// TwinCAT 3 PLC project lcls_dream_motion
// Title: lcls-dream-motion
// Company: SLAC
// ProjectVersion: 1.0.0
// ProgramVersion: 3.1.4026.17
// libraries:
//   LCLS General, * (SLAC)
//   lcls-twincat-motion, * (SLAC)
//   PMPS, * (SLAC - LCLS)
//   Tc2_MC2, * (Beckhoff Automation GmbH)
//   Tc2_Standard, * (Beckhoff Automation GmbH)
//   Tc2_System, * (Beckhoff Automation GmbH)
//   Tc3_IPCDiag, * (Beckhoff Automation GmbH)
//   Tc3_Module, * (Beckhoff Automation GmbH)
// project tree:
//   DUTs/ ENUM_AxisStates.TcDUT
//   GVLs/ GVL_EPS.TcGVL, GVL_PLC_Interfaces.TcGVL, GVL_PMPS.TcGVL, Main.TcGVL
//   / PlcTask.TcTTO
//   POUs/ PRG_SMARACT.TcPOU, PRG_CoilMovers.TcPOU, PRG_GasJetPointing.TcPOU, PRG_PLC_tasks.TcPOU, PRG_GasNozzleXYZ.TcPOU, PRG_MainChamber.TcPOU
// real-time tasks:
//   TASK PlcTask: cycle T#10ms, priority 20, ADS port 350
// motion (NC):
//   TASK NC-Task 1: cycle T#2ms, priority 4, ADS port 501
//   TASK NC- Task 1 SVB: cycle T#10ms, priority 8, ADS port 511
//   AXIS M1 -MMS-Y (id 1)
//     Dynamic: AccelerationMaximum=250, DecelerationMaximum=250, Acceleration=250, Deceleration=250, DelayTime=0.008
//     Velo: Maximum=2.5
//     OtherSettings: AllowMotionCmdToSlave=true
//     encoder EncType=29
//       EncPara: ScaleFactorNumerator=5e-05, MaxCount=#xffffffff
//         SoftEndMinControl: Range=98.55
//         SoftEndMaxControl: Range=98.73
//         Inc: RefSoftSyncMask=#x0000ffff
//     drive DrvType=24
//       Analog: VeloReferenz=2.5, ScaleFactorActTorque=0.1
//       TimeComp: TaskDelayCycles=1
//     controller CtrType=2
//       CtrPara: PriorControlFactor=1
//         PosDiffControl: Range=0.3
//         PID: PosKp=0.1, PosExtVelo=0.2, DeadBandPosition=0.1
//         Observer: BandWidth=20
//   AXIS M6_GSJN-MMS-X (id 6)
//     Dynamic: AccelerationMaximum=500, DecelerationMaximum=500, Acceleration=50, Deceleration=50, Jerk=500
//     Velo: Maximum=5
//     PositionAreaControl: Range=0.0015625
//     TargetPosControl: Range=0.0015625
//     OtherSettings: AllowMotionCmdToSlave=true
//     encoder EncType=29
//       EncPara: ScaleFactorNumerator=0.000244140625, Offset=-33543453.28, MaxCount=#xffffffff, MaxCountHighDWord=#x0000001f, ReferenceSystem=1
//         FilterTime: TVelo=0.1
//         SoftEndMinControl: Enable=true, Range=-13.5
//         SoftEndMaxControl: Enable=true, Range=11.5
//         Inc: RefSoftSyncMask=#x0000ffff
//     drive DrvType=24
//       Analog: VeloReferenz=12.5, ScaleFactorActTorque=0.1
//       TimeComp: TaskDelayCycles=1
//     controller CtrType=1
//       CtrPara: PriorControlFactor=1
//         PosDiffControl: Range=0.1
//         Observer: BandWidth=20
//   AXIS M8_GSJN-MMS-Z (id 8)
//     Dynamic: AccelerationMaximum=500, DecelerationMaximum=500, Acceleration=50, Deceleration=50, Jerk=500
//     Velo: Maximum=5
//     PositionAreaControl: Range=0.002
//     TargetPosControl: Range=0.002, Time=0.1
//     OtherSettings: AllowMotionCmdToSlave=true, NoMotionFilterTime=0.05
//     encoder EncType=29
//       EncPara: ScaleFactorNumerator=0.000244140625, Offset=-33543954.59, MaxCount=#xffffffff, MaxCountHighDWord=#x0000001f, ReferenceSystem=1
//         SoftEndMinControl: Enable=true, Range=-3.5
//         SoftEndMaxControl: Enable=true, Range=4
//         Inc: RefSoftSyncMask=#x0000ffff
//     drive DrvType=24
//       Analog: VeloReferenz=12.5, ScaleFactorActTorque=0.1
//       TimeComp: TaskDelayCycles=1
//     controller CtrType=2
//       CtrPara: PriorControlFactor=1
//         PosDiffControl: Range=0.1
//         PID: PosKp=5, PosExtKp=1, DeadBandPosition=0.001
//         Observer: BandWidth=20
//   AXIS M7_GSJN-MMS-Y (id 7)
//     Dynamic: AccelerationMaximum=500, DecelerationMaximum=500, Acceleration=50, Deceleration=50, Jerk=500
//     Velo: SlowManual=1, FastManual=2, Maximum=5.08
//     PositionAreaControl: Range=0.00127
//     TargetPosControl: Range=0.00127
//     OtherSettings: AllowMotionCmdToSlave=true, PulseDistancePos=1, PulseDistanceNeg=1
//     encoder EncType=29
//       EncPara: ScaleFactorNumerator=0.000244140625, Offset=-33550977.0786, MaxCount=#xffffffff, MaxCountHighDWord=#x0000001f, ReferenceSystem=1
//         SoftEndMinControl: Enable=true, Range=-71.06
//         SoftEndMaxControl: Enable=true, Range=0.5
//         Inc: RefSoftSyncMask=#x0000ffff
//     drive DrvType=24
//       Analog: VeloReferenz=5.08, ScaleFactorActTorque=0.1
//       TimeComp: TaskDelayCycles=1
//     controller CtrType=1
//       CtrPara: PriorControlFactor=1
//         PosDiffControl: Range=0.1
//         PID: PosKp=3
//         Observer: BandWidth=20
//   AXIS M10_DREAM_DGPD_MMT_X (id 10)
//     Dynamic: AccelerationMaximum=10, DecelerationMaximum=10, Acceleration=2.51748, Deceleration=2.51748, Jerk=9.32019
//     Velo: RefSearch=0.5, RefSync=0.4, SlowManual=0.2, FastManual=0.2, Maximum=1
//     PositionAreaControl: Range=0.005
//     TargetPosControl: Enable=false
//     OtherSettings: AllowMotionCmdToSlave=true, PulseDistancePos=0.01, PulseDistanceNeg=0.01
//     encoder EncType=19
//       EncPara: ScaleFactorNumerator=1e-06, MaxCount=#xffffffff
//     drive DrvType=16
//       DrvPara: MaxCount=#xffffffff, DriveControlDWord=#x00020100
//         Analog: VeloReferenz=1, TorqueSetpointScale=10, ScaleFactorActTorque=0.1
//         TimeComp: TaskDelayCycles=1
//     controller CtrType=1
//       CtrPara: PriorControlFactor=1
//         PosDiffControl: Range=0.05
//         Observer: BandWidth=20
//   AXIS M11_DREAM_DGPD_MMT_RET (id 11)
//     Dynamic: AccelerationMaximum=10, DecelerationMaximum=10, Acceleration=2.51748, Deceleration=2.51748, Jerk=9.32019
//     Velo: RefSearch=0.5, RefSync=0.4, SlowManual=0.2, FastManual=0.2, Maximum=1
//     PositionAreaControl: Range=0.005
//     TargetPosControl: Enable=false
//     OtherSettings: AllowMotionCmdToSlave=true, PulseDistancePos=0.01, PulseDistanceNeg=0.01
//     encoder EncType=19
//       EncPara: ScaleFactorNumerator=1e-06, MaxCount=#xffffffff
//     drive DrvType=16
//       DrvPara: MaxCount=#xffffffff, DriveControlDWord=#x00020100
//         Analog: VeloReferenz=1, TorqueSetpointScale=10, ScaleFactorActTorque=0.1
//         TimeComp: TaskDelayCycles=1
//     controller CtrType=1
//       CtrPara: PriorControlFactor=1
//         PosDiffControl: Range=0.05
//         Observer: BandWidth=20
//   AXIS M9_DREAM_DGPD_MMT_Y (id 9)
//     Dynamic: AccelerationMaximum=10, DecelerationMaximum=10, Acceleration=2.51748, Deceleration=2.51748, Jerk=9.32019
//     Velo: RefSearch=0.5, RefSync=0.4, SlowManual=0.2, FastManual=0.2, Maximum=1
//     PositionAreaControl: Range=0.005
//     TargetPosControl: Enable=false
//     OtherSettings: AllowMotionCmdToSlave=true, PulseDistancePos=0.01, PulseDistanceNeg=0.01
//     encoder EncType=19
//       EncPara: ScaleFactorNumerator=1e-06, MaxCount=#xffffffff
//     drive DrvType=16
//       DrvPara: MaxCount=#xffffffff, DriveControlDWord=#x00020100
//         Analog: VeloReferenz=1, TorqueSetpointScale=10, ScaleFactorActTorque=0.1
//         TimeComp: TaskDelayCycles=1
//     controller CtrType=1
//       CtrPara: PriorControlFactor=1
//         PosDiffControl: Range=0.05
//         Observer: BandWidth=20
//   AXIS M2 - Coil Roll (id 2)
//     Dynamic: AccelerationMaximum=1600, DecelerationMaximum=1600, Acceleration=1600, Deceleration=1600
//     Velo: Maximum=16
//     OtherSettings: AllowMotionCmdToSlave=true
//     encoder EncType=7
//       EncPara: ScaleFactorNumerator=0.004566812625, Offset=-59.42, MaxCount=#x0000ffff, ReferenceSystem=1
//         SoftEndMinControl: Enable=true, Range=-53.06
//         SoftEndMaxControl: Enable=true, Range=75.44
//         Inc: RefSoftSyncMask=#x0000ffff
//     drive DrvType=24
//       Analog: VeloReferenz=15.875, ScaleFactorActTorque=0.1
//       TimeComp: TaskDelayCycles=1
//     controller CtrType=1
//       CtrPara: PriorControlFactor=1
//         PosDiffControl: Range=1
//         Observer: BandWidth=20
//   AXIS M3 - Coil Yaw (id 3)
//     Dynamic: AccelerationMaximum=1600, DecelerationMaximum=1600
//     Velo: Maximum=16
//     OtherSettings: AllowMotionCmdToSlave=true
//     encoder EncType=7
//       EncPara: ScaleFactorNumerator=0.004566812625, Offset=-137.15, MaxCount=#x0000ffff, ReferenceSystem=1
//         SoftEndMinControl: Enable=true, Range=-3.65
//         SoftEndMaxControl: Enable=true, Range=6.35
//         Inc: RefSoftSyncMask=#x0000ffff
//     drive DrvType=24
//       Analog: VeloReferenz=15.875, ScaleFactorActTorque=0.1
//       TimeComp: TaskDelayCycles=1
//     controller CtrType=1
//       CtrPara: PriorControlFactor=1
//         PosDiffControl: Range=0.75
//         PID: PosKp=1.1
//         Observer: BandWidth=20
//   AXIS M4 - GSJP X (id 4)
//     Velo: Maximum=15.875
//     OtherSettings: AllowMotionCmdToSlave=true
//     encoder EncType=7
//       EncPara: ScaleFactorNumerator=0.0016164154, Offset=-19.9643, MaxCount=#x0000ffff, ReferenceSystem=1
//         SoftEndMinControl: Enable=true, Range=-1
//         SoftEndMaxControl: Enable=true, Range=1
//         Inc: RefSoftSyncMask=#x0000ffff
//     drive DrvType=24
//       Analog: VeloReferenz=15.875, ScaleFactorActTorque=0.1
//       TimeComp: TaskDelayCycles=1
//     controller CtrType=1
//       CtrPara: PriorControlFactor=1
//         PosDiffControl: Range=1
//         Observer: BandWidth=20
//   AXIS M5 - GSJP Z (id 5)
//     Dynamic: AccelerationMaximum=15, DecelerationMaximum=15, Acceleration=15, Deceleration=15
//     Velo: Maximum=16
//     OtherSettings: AllowMotionCmdToSlave=true
//     encoder EncType=7
//       EncPara: ScaleFactorNumerator=0.0016164154, Offset=-19.49, MaxCount=#x0000ffff, ReferenceSystem=1
//         SoftEndMinControl: Enable=true, Range=-1
//         SoftEndMaxControl: Enable=true, Range=1
//         Inc: RefSoftSyncMask=#x0000ffff
//     drive DrvType=24
//       DrvPara: Inverse=true
//         Analog: VeloReferenz=15.875, ScaleFactorActTorque=0.1
//         TimeComp: TaskDelayCycles=1
//     controller CtrType=1
//       CtrPara: PriorControlFactor=1
//         PosDiffControl: Range=1.5
//         Observer: BandWidth=20
// I/O:
//   DEVICE Device 1 (EtherCAT), AmsNetId 172.21.132.145.2.1
//     B940_009_R19_DRL_02_E0_EK1200 [EK1200-5000 EtherCAT Power supply (2A E-Bus)]
//       R19_DRL_02_EL2202
//       R19_DRL_02_E2_EL6070
//       R19_DRL_02_E3_EL6695 [EL6695 EtherCAT Bridge terminal (Primary)]
//       R19_DRL_02_E4_EK1122 [EK1122 2 port EtherCAT junction]
//         K4S08_DRL_05_E0_EK1100 [EK1100 EtherCAT Coupler (2A E-Bus)]
//           DRL_05_EL7047_E1 [EL7047 1Ch. Stepper motor output stage (50V, 5A)]
//           DRL_05_EL5042_E2 [EL5042 2Ch. BiSS-C Encoder]
//           DRL_05_EL7047_E3 [EL7047 1Ch. Stepper motor output stage (50V, 5A)]
//           DRL_05_EL7047_E4 [EL7047 1Ch. Stepper motor output stage (50V, 5A)]
//           DRL_05_EL3064_E5
//           DRL_05_EL7047_E6 [EL7047 1Ch. Stepper motor output stage (50V, 5A)]
//           DRL_05_EL7047_E7 [EL7047 1Ch. Stepper motor output stage (50V, 5A)]
//           DRL_05_EL7047_E9 [EL7047 1Ch. Stepper motor output stage (50V, 5A)]
//           DRL_05_EL7047_E10 [EL7047 1Ch. Stepper motor output stage (50V, 5A)]
//           DRL_05_EL5042_E11 [EL5042 2Ch. BiSS-C Encoder]
//           DRL_05_EL7047_E12 [EL7047 1Ch. Stepper motor output stage (50V, 5A)]
//           DRL_05_EL9011 [EL9011 End Terminal]
//         Term 35 (EK1100) [EK1100 EtherCAT Coupler (2A E-Bus)]
//           B950-100H1-R02-PNL-01_E1 [EL2624 4Ch. Relay Output, NO (125V AC / 30V DC)]
//           B950-100H1-R02-PNL-01_E2 [EL1002 2Ch. Dig. Input 24V, 3ms]
//           Term 41 (EL9011) [EL9011 End Terminal]
//         TMO-DREAM-SMARACT-03 [MCS2-3C] (disabled)
//           modules: DREAM:DGPD:MMT:Y, DREAM:DGPD:MMT:X, DREAM:DGPD:MMT:RET
//       B940_009_R19_DRL_02_E5_ EL6695 [EL6695 EtherCAT Bridge terminal (Primary)]
//       Term 42 (EL9011) [EL9011 End Terminal]
// variable links:
//   (this object) <-> Device 1 (EtherCAT)/B940_009_R19_DRL_02_E0_EK1200/R19_DRL_02_E4_EK1122/K4S08_DRL_05_E0_EK1100/DRL_05_EL5042_E2
//     Enc/Inputs/In/nComState @bit 1 <-> WcState/InputToggle
//     Enc/Inputs/In/nComState <-> WcState/WcState
//     Enc/Inputs/In/nDataIn1 <-> FB Inputs Channel 1/Position
//     Enc/Inputs/In/nDataIn1 <-> FB Inputs Channel 2/Position
//     Enc/Inputs/In/nState1 @bit 12 <-> FB Inputs Channel 1/Status/Diag
//     Enc/Inputs/In/nState1 @bit 12 <-> FB Inputs Channel 2/Status/Diag
//     Enc/Inputs/In/nState1 @bit 1 <-> FB Inputs Channel 1/Status/Error
//     Enc/Inputs/In/nState1 @bit 1 <-> FB Inputs Channel 2/Status/Error
//     Enc/Inputs/In/nState1 @bit 14 <-> FB Inputs Channel 1/Status/Input cycle counter
//     Enc/Inputs/In/nState1 @bit 14 <-> FB Inputs Channel 2/Status/Input cycle counter
//     Enc/Inputs/In/nState1 @bit 2 <-> FB Inputs Channel 1/Status/Ready
//     Enc/Inputs/In/nState1 @bit 2 <-> FB Inputs Channel 2/Status/Ready
//     Enc/Inputs/In/nState1 @bit 13 <-> FB Inputs Channel 1/Status/TxPDO State
//     Enc/Inputs/In/nState1 @bit 13 <-> FB Inputs Channel 2/Status/TxPDO State
//     Enc/Inputs/In/nState1 <-> FB Inputs Channel 1/Status/Warning
//     Enc/Inputs/In/nState1 <-> FB Inputs Channel 2/Status/Warning
//   (this object) <-> Device 1 (EtherCAT)/B940_009_R19_DRL_02_E0_EK1200/R19_DRL_02_E4_EK1122/K4S08_DRL_05_E0_EK1100/DRL_05_EL7047_E1
//     Drive/Inputs/In/nState1 @bit 3 <-> STM Status/Status/Error
//     Drive/Inputs/In/nState1 @bit 7 <-> STM Status/Status/Motor stall
//     Drive/Inputs/In/nState1 @bit 5 <-> STM Status/Status/Moving negative
//     Drive/Inputs/In/nState1 @bit 4 <-> STM Status/Status/Moving positive
//     Drive/Inputs/In/nState1 @bit 1 <-> STM Status/Status/Ready
//     Drive/Inputs/In/nState1 <-> STM Status/Status/Ready to enable
//     Drive/Inputs/In/nState1 @bit 6 <-> STM Status/Status/Torque reduced
//     Drive/Inputs/In/nState1 @bit 2 <-> STM Status/Status/Warning
//     Drive/Inputs/In/nState2 @bit 3 <-> STM Status/Status/Digital input 1
//     Drive/Inputs/In/nState2 @bit 4 <-> STM Status/Status/Digital input 2
//     Drive/Inputs/In/nState2 @bit 5 <-> STM Status/Status/Sync error
//     Drive/Inputs/In/nState2 @bit 7 <-> STM Status/Status/TxPDO Toggle
//     Drive/Inputs/In/nState4 @bit 1 <-> WcState/InputToggle
//     Drive/Inputs/In/nState4 <-> WcState/WcState
//     Drive/Outputs/Out/nCtrl1 <-> STM Control/Control/Enable
//     Drive/Outputs/Out/nCtrl1 @bit 2 <-> STM Control/Control/Reduce torque
//     Drive/Outputs/Out/nCtrl1 @bit 1 <-> STM Control/Control/Reset
//     Drive/Outputs/Out/nCtrl2 @bit 3 <-> STM Control/Control/Digital output 1
//     Drive/Outputs/Out/nDataOut2[0] <-> STM Velocity/Velocity
//   (this object) <-> Device 1 (EtherCAT)/B940_009_R19_DRL_02_E0_EK1200/R19_DRL_02_E4_EK1122/K4S08_DRL_05_E0_EK1100/DRL_05_EL7047_E9
//     Drive/Inputs/In/nState1 @bit 3 <-> STM Status/Status/Error
//     Drive/Inputs/In/nState1 @bit 7 <-> STM Status/Status/Motor stall
//     Drive/Inputs/In/nState1 @bit 5 <-> STM Status/Status/Moving negative
//     Drive/Inputs/In/nState1 @bit 4 <-> STM Status/Status/Moving positive
//     Drive/Inputs/In/nState1 @bit 1 <-> STM Status/Status/Ready
//     Drive/Inputs/In/nState1 <-> STM Status/Status/Ready to enable
//     Drive/Inputs/In/nState1 @bit 6 <-> STM Status/Status/Torque reduced
//     Drive/Inputs/In/nState1 @bit 2 <-> STM Status/Status/Warning
//     Drive/Inputs/In/nState2 @bit 3 <-> STM Status/Status/Digital input 1
//     Drive/Inputs/In/nState2 @bit 4 <-> STM Status/Status/Digital input 2
//     Drive/Inputs/In/nState2 @bit 5 <-> STM Status/Status/Sync error
//     Drive/Inputs/In/nState2 @bit 7 <-> STM Status/Status/TxPDO Toggle
//     Drive/Inputs/In/nState4 @bit 1 <-> WcState/InputToggle
//     Drive/Inputs/In/nState4 <-> WcState/WcState
//     Drive/Outputs/Out/nCtrl1 <-> STM Control/Control/Enable
//     Drive/Outputs/Out/nCtrl1 @bit 2 <-> STM Control/Control/Reduce torque
//     Drive/Outputs/Out/nCtrl1 @bit 1 <-> STM Control/Control/Reset
//     Drive/Outputs/Out/nCtrl2 @bit 3 <-> STM Control/Control/Digital output 1
//     Drive/Outputs/Out/nDataOut2[0] <-> STM Velocity/Velocity
//   (this object) <-> Device 1 (EtherCAT)/B940_009_R19_DRL_02_E0_EK1200/R19_DRL_02_E4_EK1122/K4S08_DRL_05_E0_EK1100/DRL_05_EL5042_E11
//     Enc/Inputs/In/nComState @bit 1 <-> WcState/InputToggle
//     Enc/Inputs/In/nComState <-> WcState/WcState
//     Enc/Inputs/In/nDataIn1 <-> FB Inputs Channel 2/Position
//     Enc/Inputs/In/nDataIn1 <-> FB Inputs Channel 1/Position
//     Enc/Inputs/In/nState1 @bit 12 <-> FB Inputs Channel 2/Status/Diag
//     Enc/Inputs/In/nState1 @bit 12 <-> FB Inputs Channel 1/Status/Diag
//     Enc/Inputs/In/nState1 @bit 1 <-> FB Inputs Channel 2/Status/Error
//     Enc/Inputs/In/nState1 @bit 1 <-> FB Inputs Channel 1/Status/Error
//     Enc/Inputs/In/nState1 @bit 14 <-> FB Inputs Channel 2/Status/Input cycle counter
//     Enc/Inputs/In/nState1 @bit 14 <-> FB Inputs Channel 1/Status/Input cycle counter
//     Enc/Inputs/In/nState1 @bit 2 <-> FB Inputs Channel 2/Status/Ready
//     Enc/Inputs/In/nState1 @bit 2 <-> FB Inputs Channel 1/Status/Ready
//     Enc/Inputs/In/nState1 @bit 13 <-> FB Inputs Channel 2/Status/TxPDO State
//     Enc/Inputs/In/nState1 @bit 13 <-> FB Inputs Channel 1/Status/TxPDO State
//     Enc/Inputs/In/nState1 <-> FB Inputs Channel 2/Status/Warning
//     Enc/Inputs/In/nState1 <-> FB Inputs Channel 1/Status/Warning
//   (this object) <-> Device 1 (EtherCAT)/B940_009_R19_DRL_02_E0_EK1200/R19_DRL_02_E4_EK1122/K4S08_DRL_05_E0_EK1100/DRL_05_EL7047_E12
//     Drive/Inputs/In/nState1 @bit 3 <-> STM Status/Status/Error
//     Drive/Inputs/In/nState1 @bit 7 <-> STM Status/Status/Motor stall
//     Drive/Inputs/In/nState1 @bit 5 <-> STM Status/Status/Moving negative
//     Drive/Inputs/In/nState1 @bit 4 <-> STM Status/Status/Moving positive
//     Drive/Inputs/In/nState1 @bit 1 <-> STM Status/Status/Ready
//     Drive/Inputs/In/nState1 <-> STM Status/Status/Ready to enable
//     Drive/Inputs/In/nState1 @bit 6 <-> STM Status/Status/Torque reduced
//     Drive/Inputs/In/nState1 @bit 2 <-> STM Status/Status/Warning
//     Drive/Inputs/In/nState2 @bit 3 <-> STM Status/Status/Digital input 1
//     Drive/Inputs/In/nState2 @bit 4 <-> STM Status/Status/Digital input 2
//     Drive/Inputs/In/nState2 @bit 5 <-> STM Status/Status/Sync error
//     Drive/Inputs/In/nState2 @bit 7 <-> STM Status/Status/TxPDO Toggle
//     Drive/Inputs/In/nState4 @bit 1 <-> WcState/InputToggle
//     Drive/Inputs/In/nState4 <-> WcState/WcState
//     Drive/Outputs/Out/nCtrl1 <-> STM Control/Control/Enable
//     Drive/Outputs/Out/nCtrl1 @bit 2 <-> STM Control/Control/Reduce torque
//     Drive/Outputs/Out/nCtrl1 @bit 1 <-> STM Control/Control/Reset
//     Drive/Outputs/Out/nCtrl2 @bit 3 <-> STM Control/Control/Digital output 1
//     Drive/Outputs/Out/nDataOut2[0] <-> STM Velocity/Velocity
//   (this object) <-> Device 1 (EtherCAT)/B940_009_R19_DRL_02_E0_EK1200/R19_DRL_02_E4_EK1122/K4S08_DRL_05_E0_EK1100/DRL_05_EL7047_E10
//     Drive/Inputs/In/nState1 @bit 3 <-> STM Status/Status/Error
//     Drive/Inputs/In/nState1 @bit 7 <-> STM Status/Status/Motor stall
//     Drive/Inputs/In/nState1 @bit 5 <-> STM Status/Status/Moving negative
//     Drive/Inputs/In/nState1 @bit 4 <-> STM Status/Status/Moving positive
//     Drive/Inputs/In/nState1 @bit 1 <-> STM Status/Status/Ready
//     Drive/Inputs/In/nState1 <-> STM Status/Status/Ready to enable
//     Drive/Inputs/In/nState1 @bit 6 <-> STM Status/Status/Torque reduced
//     Drive/Inputs/In/nState1 @bit 2 <-> STM Status/Status/Warning
//     Drive/Inputs/In/nState2 @bit 3 <-> STM Status/Status/Digital input 1
//     Drive/Inputs/In/nState2 @bit 4 <-> STM Status/Status/Digital input 2
//     Drive/Inputs/In/nState2 @bit 5 <-> STM Status/Status/Sync error
//     Drive/Inputs/In/nState2 @bit 7 <-> STM Status/Status/TxPDO Toggle
//     Drive/Inputs/In/nState4 @bit 1 <-> WcState/InputToggle
//     Drive/Inputs/In/nState4 <-> WcState/WcState
//     Drive/Outputs/Out/nCtrl1 <-> STM Control/Control/Enable
//     Drive/Outputs/Out/nCtrl1 @bit 2 <-> STM Control/Control/Reduce torque
//     Drive/Outputs/Out/nCtrl1 @bit 1 <-> STM Control/Control/Reset
//     Drive/Outputs/Out/nCtrl2 @bit 3 <-> STM Control/Control/Digital output 1
//     Drive/Outputs/Out/nDataOut2[0] <-> STM Velocity/Velocity
//   (this object) <-> Device 1 (EtherCAT)/B940_009_R19_DRL_02_E0_EK1200/R19_DRL_02_E4_EK1122/TMO-DREAM-SMARACT-03
//     Drive/Inputs/In/nDataIn1 <-> DREAM:DGPD:MMT:X/mode/status/pos/fError TxPDO/Following Error Actual Value
//     Drive/Inputs/In/nState1 <-> DREAM:DGPD:MMT:X/mode/status/pos/fError TxPDO/Status Word
//     Drive/Inputs/In/nState2 <-> DREAM:DGPD:MMT:X/mode/status/pos/fError TxPDO/Status Word @bit 8
//     Drive/Inputs/In/nState4 @bit 1 <-> WcState/InputToggle
//     Drive/Inputs/In/nState4 <-> WcState/WcState
//     Drive/Inputs/In/nState5 <-> DREAM:DGPD:MMT:X/mode/status/pos/fError TxPDO/Modes of Operation Display
//     Drive/Outputs/Out/nDataOut1 <-> DREAM:DGPD:MMT:X/ctl/mode/pos RxPDO/Target Position
//     Enc/Inputs/In/nDataIn1 <-> DREAM:DGPD:MMT:X/mode/status/pos/fError TxPDO/Position Actual Value
//     Enc/Inputs/In/nState4 @bit 1 <-> WcState/InputToggle
//     Enc/Inputs/In/nState4 <-> WcState/WcState
//     Drive/Inputs/In/nDataIn1 <-> DREAM:DGPD:MMT:RET/mode/status/pos/fError TxPDO/Following Error Actual Value
//     Drive/Inputs/In/nState1 <-> DREAM:DGPD:MMT:RET/mode/status/pos/fError TxPDO/Status Word
//     Drive/Inputs/In/nState2 <-> DREAM:DGPD:MMT:RET/mode/status/pos/fError TxPDO/Status Word @bit 8
//     Drive/Inputs/In/nState5 <-> DREAM:DGPD:MMT:RET/mode/status/pos/fError TxPDO/Modes of Operation Display
//     Drive/Outputs/Out/nDataOut1 <-> DREAM:DGPD:MMT:RET/ctl/mode/pos RxPDO/Target Position
//     Enc/Inputs/In/nDataIn1 <-> DREAM:DGPD:MMT:RET/mode/status/pos/fError TxPDO/Position Actual Value
//     Drive/Inputs/In/nDataIn1 <-> DREAM:DGPD:MMT:Y/mode/status/pos/fError TxPDO/Following Error Actual Value
//     Drive/Inputs/In/nState1 <-> DREAM:DGPD:MMT:Y/mode/status/pos/fError TxPDO/Status Word
//     Drive/Inputs/In/nState2 <-> DREAM:DGPD:MMT:Y/mode/status/pos/fError TxPDO/Status Word @bit 8
//     Drive/Inputs/In/nState5 <-> DREAM:DGPD:MMT:Y/mode/status/pos/fError TxPDO/Modes of Operation Display
//     Drive/Outputs/Out/nDataOut1 <-> DREAM:DGPD:MMT:Y/ctl/mode/pos RxPDO/Target Position
//     Enc/Inputs/In/nDataIn1 <-> DREAM:DGPD:MMT:Y/mode/status/pos/fError TxPDO/Position Actual Value
//   (this object) <-> Device 1 (EtherCAT)/B940_009_R19_DRL_02_E0_EK1200/R19_DRL_02_E4_EK1122/K4S08_DRL_05_E0_EK1100/DRL_05_EL3064_E5
//     Enc/Inputs/In/nDataIn1[0] <-> AI Standard Channel {1..4}/Value  (4 links)
//     Enc/Inputs/In/nState4 @bit 1 <-> WcState/InputToggle
//     Enc/Inputs/In/nState4 <-> WcState/WcState
//   (this object) <-> Device 1 (EtherCAT)/B940_009_R19_DRL_02_E0_EK1200/R19_DRL_02_E4_EK1122/K4S08_DRL_05_E0_EK1100/DRL_05_EL7047_E3
//     Drive/Inputs/In/nState1 @bit 3 <-> STM Status/Status/Error
//     Drive/Inputs/In/nState1 @bit 7 <-> STM Status/Status/Motor stall
//     Drive/Inputs/In/nState1 @bit 5 <-> STM Status/Status/Moving negative
//     Drive/Inputs/In/nState1 @bit 4 <-> STM Status/Status/Moving positive
//     Drive/Inputs/In/nState1 @bit 1 <-> STM Status/Status/Ready
//     Drive/Inputs/In/nState1 <-> STM Status/Status/Ready to enable
//     Drive/Inputs/In/nState1 @bit 6 <-> STM Status/Status/Torque reduced
//     Drive/Inputs/In/nState1 @bit 2 <-> STM Status/Status/Warning
//     Drive/Inputs/In/nState2 @bit 3 <-> STM Status/Status/Digital input 1
//     Drive/Inputs/In/nState2 @bit 4 <-> STM Status/Status/Digital input 2
//     Drive/Inputs/In/nState2 @bit 5 <-> STM Status/Status/Sync error
//     Drive/Inputs/In/nState2 @bit 7 <-> STM Status/Status/TxPDO Toggle
//     Drive/Inputs/In/nState4 @bit 1 <-> WcState/InputToggle
//     Drive/Inputs/In/nState4 <-> WcState/WcState
//     Drive/Outputs/Out/nCtrl1 <-> STM Control/Control/Enable
//     Drive/Outputs/Out/nCtrl1 @bit 2 <-> STM Control/Control/Reduce torque
//     Drive/Outputs/Out/nCtrl1 @bit 1 <-> STM Control/Control/Reset
//     Drive/Outputs/Out/nCtrl2 @bit 3 <-> STM Control/Control/Digital output 1
//     Drive/Outputs/Out/nDataOut2[0] <-> STM Velocity/Velocity
//   (this object) <-> Device 1 (EtherCAT)/B940_009_R19_DRL_02_E0_EK1200/R19_DRL_02_E4_EK1122/K4S08_DRL_05_E0_EK1100/DRL_05_EL7047_E4
//     Drive/Inputs/In/nState1 @bit 3 <-> STM Status/Status/Error
//     Drive/Inputs/In/nState1 @bit 7 <-> STM Status/Status/Motor stall
//     Drive/Inputs/In/nState1 @bit 5 <-> STM Status/Status/Moving negative
//     Drive/Inputs/In/nState1 @bit 4 <-> STM Status/Status/Moving positive
//     Drive/Inputs/In/nState1 @bit 1 <-> STM Status/Status/Ready
//     Drive/Inputs/In/nState1 <-> STM Status/Status/Ready to enable
//     Drive/Inputs/In/nState1 @bit 6 <-> STM Status/Status/Torque reduced
//     Drive/Inputs/In/nState1 @bit 2 <-> STM Status/Status/Warning
//     Drive/Inputs/In/nState2 @bit 3 <-> STM Status/Status/Digital input 1
//     Drive/Inputs/In/nState2 @bit 4 <-> STM Status/Status/Digital input 2
//     Drive/Inputs/In/nState2 @bit 5 <-> STM Status/Status/Sync error
//     Drive/Inputs/In/nState2 @bit 7 <-> STM Status/Status/TxPDO Toggle
//     Drive/Inputs/In/nState4 @bit 1 <-> WcState/InputToggle
//     Drive/Inputs/In/nState4 <-> WcState/WcState
//     Drive/Outputs/Out/nCtrl1 <-> STM Control/Control/Enable
//     Drive/Outputs/Out/nCtrl1 @bit 2 <-> STM Control/Control/Reduce torque
//     Drive/Outputs/Out/nCtrl1 @bit 1 <-> STM Control/Control/Reset
//     Drive/Outputs/Out/nCtrl2 @bit 3 <-> STM Control/Control/Digital output 1
//     Drive/Outputs/Out/nDataOut2[0] <-> STM Velocity/Velocity
//   (this object) <-> Device 1 (EtherCAT)/B940_009_R19_DRL_02_E0_EK1200/R19_DRL_02_E4_EK1122/K4S08_DRL_05_E0_EK1100/DRL_05_EL7047_E6
//     Drive/Inputs/In/nState1 @bit 3 <-> STM Status/Status/Error
//     Drive/Inputs/In/nState1 @bit 7 <-> STM Status/Status/Motor stall
//     Drive/Inputs/In/nState1 @bit 5 <-> STM Status/Status/Moving negative
//     Drive/Inputs/In/nState1 @bit 4 <-> STM Status/Status/Moving positive
//     Drive/Inputs/In/nState1 @bit 1 <-> STM Status/Status/Ready
//     Drive/Inputs/In/nState1 <-> STM Status/Status/Ready to enable
//     Drive/Inputs/In/nState1 @bit 6 <-> STM Status/Status/Torque reduced
//     Drive/Inputs/In/nState1 @bit 2 <-> STM Status/Status/Warning
//     Drive/Inputs/In/nState2 @bit 3 <-> STM Status/Status/Digital input 1
//     Drive/Inputs/In/nState2 @bit 4 <-> STM Status/Status/Digital input 2
//     Drive/Inputs/In/nState2 @bit 5 <-> STM Status/Status/Sync error
//     Drive/Inputs/In/nState2 @bit 7 <-> STM Status/Status/TxPDO Toggle
//     Drive/Inputs/In/nState4 @bit 1 <-> WcState/InputToggle
//     Drive/Inputs/In/nState4 <-> WcState/WcState
//     Drive/Outputs/Out/nCtrl1 <-> STM Control/Control/Enable
//     Drive/Outputs/Out/nCtrl1 @bit 2 <-> STM Control/Control/Reduce torque
//     Drive/Outputs/Out/nCtrl1 @bit 1 <-> STM Control/Control/Reset
//     Drive/Outputs/Out/nCtrl2 @bit 3 <-> STM Control/Control/Digital output 1
//     Drive/Outputs/Out/nDataOut2[0] <-> STM Velocity/Velocity
//   (this object) <-> Device 1 (EtherCAT)/B940_009_R19_DRL_02_E0_EK1200/R19_DRL_02_E4_EK1122/K4S08_DRL_05_E0_EK1100/DRL_05_EL7047_E7
//     Drive/Inputs/In/nState1 @bit 3 <-> STM Status/Status/Error
//     Drive/Inputs/In/nState1 @bit 7 <-> STM Status/Status/Motor stall
//     Drive/Inputs/In/nState1 @bit 5 <-> STM Status/Status/Moving negative
//     Drive/Inputs/In/nState1 @bit 4 <-> STM Status/Status/Moving positive
//     Drive/Inputs/In/nState1 @bit 1 <-> STM Status/Status/Ready
//     Drive/Inputs/In/nState1 <-> STM Status/Status/Ready to enable
//     Drive/Inputs/In/nState1 @bit 6 <-> STM Status/Status/Torque reduced
//     Drive/Inputs/In/nState1 @bit 2 <-> STM Status/Status/Warning
//     Drive/Inputs/In/nState2 @bit 3 <-> STM Status/Status/Digital input 1
//     Drive/Inputs/In/nState2 @bit 4 <-> STM Status/Status/Digital input 2
//     Drive/Inputs/In/nState2 @bit 5 <-> STM Status/Status/Sync error
//     Drive/Inputs/In/nState2 @bit 7 <-> STM Status/Status/TxPDO Toggle
//     Drive/Inputs/In/nState4 @bit 1 <-> WcState/InputToggle
//     Drive/Inputs/In/nState4 <-> WcState/WcState
//     Drive/Outputs/Out/nCtrl1 <-> STM Control/Control/Enable
//     Drive/Outputs/Out/nCtrl1 @bit 2 <-> STM Control/Control/Reduce torque
//     Drive/Outputs/Out/nCtrl1 @bit 1 <-> STM Control/Control/Reset
//     Drive/Outputs/Out/nCtrl2 @bit 3 <-> STM Control/Control/Digital output 1
//     Drive/Outputs/Out/nDataOut2[0] <-> STM Velocity/Velocity
//   lcls_dream_motion Instance <-> Device 1 (EtherCAT)/B940_009_R19_DRL_02_E0_EK1200/R19_DRL_02_E4_EK1122/K4S08_DRL_05_E0_EK1100/DRL_05_EL3064_E5
//     PlcTask Inputs/Main.M{2..5}.nRawEncoderINT <-> AI Standard Channel {1..4}/Value  (4 links)
//   lcls_dream_motion Instance <-> Device 1 (EtherCAT)/B940_009_R19_DRL_02_E0_EK1200/R19_DRL_02_E4_EK1122/K4S08_DRL_05_E0_EK1100/DRL_05_EL5042_E11
//     PlcTask Inputs/Main.M7.nRawEncoderULINT <-> FB Inputs Channel 1/Position
//     PlcTask Inputs/Main.M8.nRawEncoderULINT <-> FB Inputs Channel 2/Position
//   lcls_dream_motion Instance <-> Device 1 (EtherCAT)/B940_009_R19_DRL_02_E0_EK1200/R19_DRL_02_E4_EK1122/K4S08_DRL_05_E0_EK1100/DRL_05_EL5042_E2
//     PlcTask Inputs/Main.M1.nRawEncoderULINT <-> FB Inputs Channel 1/Position
//     PlcTask Inputs/Main.M6.nRawEncoderULINT <-> FB Inputs Channel 2/Position
//   lcls_dream_motion Instance <-> Device 1 (EtherCAT)/B940_009_R19_DRL_02_E0_EK1200/R19_DRL_02_E4_EK1122/K4S08_DRL_05_E0_EK1100/DRL_05_EL7047_E1
//     PlcTask Inputs/Main.M1.bLimitBackwardEnable <-> STM Status/Status/Digital input 2
//     PlcTask Inputs/Main.M1.bLimitForwardEnable <-> STM Status/Status/Digital input 1
//   lcls_dream_motion Instance <-> Device 1 (EtherCAT)/B940_009_R19_DRL_02_E0_EK1200/R19_DRL_02_E4_EK1122/K4S08_DRL_05_E0_EK1100/DRL_05_EL7047_E10
//     PlcTask Inputs/Main.M7.bLimitBackwardEnable <-> STM Status/Status/Digital input 1
//     PlcTask Inputs/Main.M7.bLimitForwardEnable <-> STM Status/Status/Digital input 2
//   lcls_dream_motion Instance <-> Device 1 (EtherCAT)/B940_009_R19_DRL_02_E0_EK1200/R19_DRL_02_E4_EK1122/K4S08_DRL_05_E0_EK1100/DRL_05_EL7047_E12
//     PlcTask Inputs/Main.M8.bLimitBackwardEnable <-> STM Status/Status/Digital input 1
//     PlcTask Inputs/Main.M8.bLimitForwardEnable <-> STM Status/Status/Digital input 2
//   lcls_dream_motion Instance <-> Device 1 (EtherCAT)/B940_009_R19_DRL_02_E0_EK1200/R19_DRL_02_E4_EK1122/K4S08_DRL_05_E0_EK1100/DRL_05_EL7047_E3
//     PlcTask Inputs/Main.M2.bLimitBackwardEnable <-> STM Status/Status/Digital input 2
//     PlcTask Inputs/Main.M2.bLimitForwardEnable <-> STM Status/Status/Digital input 1
//   lcls_dream_motion Instance <-> Device 1 (EtherCAT)/B940_009_R19_DRL_02_E0_EK1200/R19_DRL_02_E4_EK1122/K4S08_DRL_05_E0_EK1100/DRL_05_EL7047_E4
//     PlcTask Inputs/Main.M3.bLimitBackwardEnable <-> STM Status/Status/Digital input 2
//     PlcTask Inputs/Main.M3.bLimitForwardEnable <-> STM Status/Status/Digital input 1
//   lcls_dream_motion Instance <-> Device 1 (EtherCAT)/B940_009_R19_DRL_02_E0_EK1200/R19_DRL_02_E4_EK1122/K4S08_DRL_05_E0_EK1100/DRL_05_EL7047_E6
//     PlcTask Inputs/Main.M4.bLimitBackwardEnable <-> STM Status/Status/Digital input 2
//     PlcTask Inputs/Main.M4.bLimitForwardEnable <-> STM Status/Status/Digital input 1
//   lcls_dream_motion Instance <-> Device 1 (EtherCAT)/B940_009_R19_DRL_02_E0_EK1200/R19_DRL_02_E4_EK1122/K4S08_DRL_05_E0_EK1100/DRL_05_EL7047_E7
//     PlcTask Inputs/Main.M5.bLimitBackwardEnable <-> STM Status/Status/Digital input 1
//     PlcTask Inputs/Main.M5.bLimitForwardEnable <-> STM Status/Status/Digital input 2
//   lcls_dream_motion Instance <-> Device 1 (EtherCAT)/B940_009_R19_DRL_02_E0_EK1200/R19_DRL_02_E4_EK1122/K4S08_DRL_05_E0_EK1100/DRL_05_EL7047_E9
//     PlcTask Inputs/Main.M6.bLimitBackwardEnable <-> STM Status/Status/Digital input 1
//     PlcTask Inputs/Main.M6.bLimitForwardEnable <-> STM Status/Status/Digital input 2
//   lcls_dream_motion Instance <-> NC-Task 1/Axes/M1 -MMS-Y
//     PlcTask Inputs/Main.M1.Axis.NcToPlc <-> Outputs/ToPlc
//     PlcTask Outputs/Main.M1.Axis.PlcToNc <-> Inputs/FromPlc
//   lcls_dream_motion Instance <-> NC-Task 1/Axes/M2 - Coil Roll
//     PlcTask Inputs/Main.M2.Axis.NcToPlc <-> Outputs/ToPlc
//     PlcTask Outputs/Main.M2.Axis.PlcToNc <-> Inputs/FromPlc
//   lcls_dream_motion Instance <-> NC-Task 1/Axes/M3 - Coil Yaw
//     PlcTask Inputs/Main.M3.Axis.NcToPlc <-> Outputs/ToPlc
//     PlcTask Outputs/Main.M3.Axis.PlcToNc <-> Inputs/FromPlc
//   lcls_dream_motion Instance <-> NC-Task 1/Axes/M4 - GSJP X
//     PlcTask Inputs/Main.M4.Axis.NcToPlc <-> Outputs/ToPlc
//     PlcTask Outputs/Main.M4.Axis.PlcToNc <-> Inputs/FromPlc
//   lcls_dream_motion Instance <-> NC-Task 1/Axes/M5 - GSJP Z
//     PlcTask Inputs/Main.M5.Axis.NcToPlc <-> Outputs/ToPlc
//     PlcTask Outputs/Main.M5.Axis.PlcToNc <-> Inputs/FromPlc
//   lcls_dream_motion Instance <-> NC-Task 1/Axes/M6_GSJN-MMS-X
//     PlcTask Inputs/Main.M6.Axis.NcToPlc <-> Outputs/ToPlc
//     PlcTask Outputs/Main.M6.Axis.PlcToNc <-> Inputs/FromPlc
//   lcls_dream_motion Instance <-> NC-Task 1/Axes/M7_GSJN-MMS-Y
//     PlcTask Inputs/Main.M7.Axis.NcToPlc <-> Outputs/ToPlc
//     PlcTask Outputs/Main.M7.Axis.PlcToNc <-> Inputs/FromPlc
//   lcls_dream_motion Instance <-> NC-Task 1/Axes/M8_GSJN-MMS-Z
//     PlcTask Inputs/Main.M8.Axis.NcToPlc <-> Outputs/ToPlc
//     PlcTask Outputs/Main.M8.Axis.PlcToNc <-> Inputs/FromPlc

CONFIGURATION lcls_dream_motion
    RESOURCE PLC ON TwinCAT3
        TASK PlcTask(INTERVAL := T#10ms, PRIORITY := 20);
        PROGRAM PRG_PLC_tasks WITH PlcTask : PRG_PLC_tasks;
    END_RESOURCE
END_CONFIGURATION

// ---- DUTs/ENUM_AxisStates.TcDUT
{attribute 'qualified_only'}
{attribute 'strict'}
{attribute 'to_string'}
TYPE ENUM_AxisStates :
(
    UNKNOWN := 0, // UNKNOWN must be in slot 0 or the FB breaks
    OUT := 1,
    SI3N4 := 2,
    FR_YAG := 3,
    CL_YAG := 4,
    OPEN := 5,
    SMA := 6
) UINT;
END_TYPE

// ---- GVLs/GVL_EPS.TcGVL
{attribute 'qualified_only'}
VAR_GLOBAL
	(*
	{attribute 'TcLinkTo' := 'TIID^Device 1 (EtherCAT)^B940_009_R19_DRL_02_E0_EK1200^R19_DRL_02_E4_EK1122^Term 35 (EK1100)^B950-100H1-R02-PNL-01_E2^Channel 1^Input'}
    {attribute 'pytmc' := '
        pv: "DREAM:SL:STATUS",
        field: "DREAM Safety Loop Status",
        field: "ZNAM OPEN",
        field: "ONAM CLOSED"
    '}
    bSafetyLoopStatus AT %I* : BOOL;

	{attribute 'TcLinkTo' := 'TIID^Device 1 (EtherCAT)^B940_009_R19_DRL_02_E0_EK1200^R19_DRL_02_E4_EK1122^Term 35 (EK1100)^B950-100H1-R02-PNL-01_E1^Channel 1^Output'}
    {attribute 'pytmc' := '
        pv: "DREAM:SL:ENABLE",
        field: "DREAM Safety Loop Enable",
        field: "ZNAM OPEN",
        field: "ONAM CLOSED"
    '}
    bSafetyLoopEnable AT %Q*: BOOL;
	*)
END_VAR

// ---- GVLs/GVL_PLC_Interfaces.TcGVL
//{attribute 'qualified_only'}
VAR_GLOBAL
    (*ETHERCAT BRRIDGE COM STATUS*)
    //0: Other side is in OP state, >0: Error
    {attribute 'TcLinkTo' := 'TIIB[R19_DRL_02_E3_EL6695]^SYNC Inputs^TxPDO state
    '}
    xEcatBridge_TxPDO_state AT %I* :BOOL;

    //0: External device connectd, 1: External device not connected

    {attribute := 'TIIB[R19_DRL_02_E3_EL6695]^SYNC Inputs^External device not connected
    '}
    xEcatBridge_External_device_not_connected AT %I* : BOOL;

    //0 = Data valid, 1 = Data invalid
    {attribute 'TcLinkTo' := 'TIIB[R19_DRL_02_E3_EL6695]^WcState^WcState
    '}
    xEcatBridge_WcState AT %I* : BOOL;

    {attribute 'TcLinkTo' := 'TIIB[R19_DRL_02_E3_EL6695]^IO Inputs^DREAM_VRC_DP1_OPEN_LS'}
    bDREAM_VRC_DP1_OPEN_LS  AT %I* : BOOL;

    {attribute  'TcLinkTo' := 'TIIB[R19_DRL_02_E3_EL6695]^IO Outputs^DREAM_GNZ_Y_OUT'}
    xDREAM_GNZ_Y_OUT AT %Q*: BOOL;

    {attribute  'TcLinkTo' := 'TIIB[R19_DRL_02_E3_EL6695]^IO Outputs^DREAM_GNZ_Y_Ext_OUT'}
    xDREAM_GNZ_Y_Ext_OUT AT %Q*: BOOL;
END_VAR

// ---- GVLs/GVL_PMPS.TcGVL
{attribute 'qualified_only'}
VAR_GLOBAL
    (*
    {attribute 'pytmc' := 'pv: DREAM:MOTION:ARB:01'}
    fbArbiter1: FB_Arbiter(1);

    {attribute 'pytmc' := 'pv: DREAM:MOTION:FFO:02'}
    fbFastFaultOutput1: FB_HardwareFFOutput := (bAutoReset := TRUE, i_sNetID:='172.21.92.73.1.1');
    *)
END_VAR

// ---- GVLs/Main.TcGVL
{attribute 'qualified_only'}
VAR_GLOBAL
    {attribute 'pytmc' := 'pv: DREAM:MC:MMS:Y '}
    {attribute 'TcLinkTo' := '.bLimitForwardEnable  := TIIB[DRL_05_EL7047_E1]^STM Status^Status^Digital input 1;
                              .bLimitBackwardEnable := TIIB[DRL_05_EL7047_E1]^STM Status^Status^Digital input 2;
                              .nRawEncoderULINT     := TIIB[DRL_05_EL5042_E2]^FB Inputs Channel 1^Position'}
    M1: ST_MotionStage := (sName := 'DREAM:MC:MMS:Y ');

    {attribute 'pytmc' := 'pv: DREAM:COIL:MMS:ROLL '}
    {attribute 'TcLinkTo' := '.bLimitForwardEnable  := TIIB[DRL_05_EL7047_E3]^STM Status^Status^Digital input 1;
                              .bLimitBackwardEnable := TIIB[DRL_05_EL7047_E3]^STM Status^Status^Digital input 2;
                              .nRawEncoderINT     := TIIB[DRL_05_EL3064_E5]^AI Standard Channel 1^Value'}
    M2: ST_MotionStage := (sName := 'DREAM:COIL:MMS:ROLL ');

    {attribute 'pytmc' := 'pv: DREAM:COIL:MMS:YAW '}
    {attribute 'TcLinkTo' := '.bLimitForwardEnable  := TIIB[DRL_05_EL7047_E4]^STM Status^Status^Digital input 1;
                              .bLimitBackwardEnable := TIIB[DRL_05_EL7047_E4]^STM Status^Status^Digital input 2;
                              .nRawEncoderINT     := TIIB[DRL_05_EL3064_E5]^AI Standard Channel 2^Value'}
    M3: ST_MotionStage := (sName := 'DREAM:COIL:MMS:YAW ');

    {attribute 'pytmc' := 'pv: DREAM:GSJP:MMS:X '}
    {attribute 'TcLinkTo' := '.bLimitForwardEnable  := TIIB[DRL_05_EL7047_E6]^STM Status^Status^Digital input 1;
                              .bLimitBackwardEnable := TIIB[DRL_05_EL7047_E6]^STM Status^Status^Digital input 2;
                              .nRawEncoderINT     := TIIB[DRL_05_EL3064_E5]^AI Standard Channel 3^Value'}
    M4: ST_MotionStage := (sName := 'DREAM:GSJP:MMS:X ');

    {attribute 'pytmc' := 'pv: DREAM:GSJP:MMS:Z '}
    {attribute 'TcLinkTo' := '.bLimitForwardEnable  := TIIB[DRL_05_EL7047_E7]^STM Status^Status^Digital input 2;
                              .bLimitBackwardEnable := TIIB[DRL_05_EL7047_E7]^STM Status^Status^Digital input 1;
                              .nRawEncoderINT     := TIIB[DRL_05_EL3064_E5]^AI Standard Channel 4^Value'}
    M5: ST_MotionStage := (sName := 'DREAM:GSJP:MMS:Z ');

    {attribute 'pytmc' := 'pv: DREAM:GSJN:MMS:X'}
    {attribute 'TcLinkTo' := '.bLimitForwardEnable  := TIIB[DRL_05_EL7047_E9]^STM Status^Status^Digital input 2;
                              .bLimitBackwardEnable := TIIB[DRL_05_EL7047_E9]^STM Status^Status^Digital input 1;
                              .nRawEncoderULINT     := TIIB[DRL_05_EL5042_E2]^FB Inputs Channel 2^Position'}
    M6: ST_MotionStage := (sName := 'DREAM:GSJN:MMS:X');

    {attribute 'pytmc' := 'pv: DREAM:GSJN:MMS:Y'}
    {attribute 'TcLinkTo' := '.bLimitForwardEnable  := TIIB[DRL_05_EL7047_E10]^STM Status^Status^Digital input 2;
                              .bLimitBackwardEnable := TIIB[DRL_05_EL7047_E10]^STM Status^Status^Digital input 1;
                              .nRawEncoderULINT     := TIIB[DRL_05_EL5042_E11]^FB Inputs Channel 1^Position'}
    M7: ST_MotionStage := (sName := 'DREAM:GSJN:MMS:Y');

    {attribute 'pytmc' := 'pv: DREAM:GSJN:MMS:Z'}
    {attribute 'TcLinkTo' := '.bLimitForwardEnable  := TIIB[DRL_05_EL7047_E12]^STM Status^Status^Digital input 2;
                              .bLimitBackwardEnable := TIIB[DRL_05_EL7047_E12]^STM Status^Status^Digital input 1;
                              .nRawEncoderULINT     := TIIB[DRL_05_EL5042_E11]^FB Inputs Channel 2^Position'}
    M8: ST_MotionStage := (sName := 'DREAM:GSJN:MMS:Z');
	
	// In-Vacuum Motion
	(*
    {attribute 'pytmc':='pv: DREAM:DGPD:MMT:Y'}
    {attribute 'TcLinkTo' := '
        .nRawEncoderDINT		:=TIID^Device 1 (EtherCAT)^B940_009_R19_DRL_02_E0_EK1200^R19_DRL_02_E4_EK1122^TMO-DREAM-SMARACT-03^DREAM:DGPD:MMT:Y^mode/status/pos/fError TxPDO^Position Actual Value
    '}
    M9 : ST_MotionStage := (sName:='DREAM:DGPD:MMT:Y',
							nHomingMode:=E_EpicsHomeCmd.NONE,
                            // NB: Must be this 'DURING_MOTION'
							nEnableMode:= ENUM_StageEnableMode.DURING_MOTION,
							bPowerSelf:=TRUE,
							bHardwareEnable:=TRUE );

	////
	{attribute 'pytmc':='pv: DREAM:DGPD:MMT:X'}
    {attribute 'TcLinkTo' := '
        .nRawEncoderDINT		:=TIID^Device 1 (EtherCAT)^B940_009_R19_DRL_02_E0_EK1200^R19_DRL_02_E4_EK1122^TMO-DREAM-SMARACT-03^DREAM:DGPD:MMT:X^mode/status/pos/fError TxPDO^Position Actual Value
    '}
    M10 : ST_MotionStage := (sName:='DREAM:DGPD:MMT:X',
                             nHomingMode:=E_EpicsHomeCmd.NONE,
                             // NB: Must be this 'DURING_MOTION'
                             nEnableMode:= ENUM_StageEnableMode.DURING_MOTION,
                             bPowerSelf:=TRUE,
                             bHardwareEnable:=TRUE );
	////
	{attribute 'pytmc':='pv: DREAM:DGPD:MMT:RET'}
    {attribute 'TcLinkTo' := '
        .nRawEncoderDINT		:=TIID^Device 1 (EtherCAT)^B940_009_R19_DRL_02_E0_EK1200^R19_DRL_02_E4_EK1122^TMO-DREAM-SMARACT-03^DREAM:DGPD:MMT:RET^mode/status/pos/fError TxPDO^Position Actual Value
    '}
    M11 : ST_MotionStage := (	sName:='DREAM:DGPD:MMT:RET',
                                nHomingMode:=E_EpicsHomeCmd.NONE,
                                // NB: Must be this 'DURING_MOTION'
                                nEnableMode:= ENUM_StageEnableMode.DURING_MOTION,
                                bPowerSelf:=TRUE,
                                bHardwareEnable:=TRUE );
	*)						
END_VAR

// ---- POUs/PRG_PLC_tasks.TcPOU
PROGRAM PRG_PLC_tasks
VAR
    // variables for testing
    axis: AXIS_REF;
    power: MC_POWER;

    retractedLS AT %I* : BOOL;
    extendedLS At %I* :BOOL;

END_VAR


(*
   This is to test axis safely by both limit switch enabled.
   manually link the variables "retractedLS" and "extendedLS" to the imit switches inputs

   Standard limit switches are NC, enable/disable both directions directly by limit switches
  if limit swithes are NO, enable/disable the related direction using reversed limit switch reading.

*)
power(Axis:=axis, Enable_Positive := retractedLS and extendedLS, Enable_Negative:= extendedLS and retractedLS);
//power(Axis:=axis, Enable_Positive := NOT retractedLS, Enable_Negative:= NOT extendedLS);

PRG_GasNozzleXYZ();
PRG_MainChamber();
PRG_GasJetPointing();
PRG_CoilMovers();
// PRG_SMARACT();

END_PROGRAM

// ---- POUs/PRG_GasNozzleXYZ.TcPOU
PROGRAM PRG_GasNozzleXYZ
VAR
    fb_GSJN_X : FB_MotionStage;
    fb_GSJN_Y : FB_MotionStage;
    fb_GSJN_Z : FB_MotionStage;

    bInit : BOOl := TRUE;

END_VAR

IF ( bInit) THEN
    bInit := FALSE;
    Main.M6.bHardwareEnable := TRUE;
    Main.M6.bPowerSelf := TRUE;
    Main.M6.fVelocity := 0.05;
    Main.M6.nBrakeMode := ENUM_StageBrakeMode.NO_BRAKE;
    Main.M6.nEnableMode := ENUM_StageEnableMode.DURING_MOTION;

    Main.M7.bHardwareEnable := TRUE;
    Main.M7.bPowerSelf := TRUE;
    Main.M7.fVelocity := 0.05;
    Main.M7.nBrakeMode := ENUM_StageBrakeMode.NO_BRAKE;
    Main.M7.nEnableMode := ENUM_StageEnableMode.DURING_MOTION;

    Main.M8.bHardwareEnable := TRUE;
    Main.M8.bPowerSelf := TRUE;
    Main.M8.fVelocity := 0.05;
    Main.M8.nBrakeMode := ENUM_StageBrakeMode.NO_BRAKE;
    Main.M8.nEnableMode := ENUM_StageEnableMode.DURING_MOTION;
END_IF

fb_GSJN_X(stMotionStage:=Main.M6);
fb_GSJN_Y(stMotionStage:=Main.M7);
fb_GSJN_Z(stMotionStage:=Main.M8);

END_PROGRAM

// ---- POUs/PRG_MainChamber.TcPOU
PROGRAM PRG_MainChamber
VAR
    fb_MC_Y : FB_MotionStage;
    bInit : BOOL := TRUE;
END_VAR

IF ( bInit) THEN
    bInit := FALSE;
    Main.M1.bHardwareEnable := TRUE;
    Main.M1.bPowerSelf := TRUE;
    Main.M1.nBrakeMode := ENUM_StageBrakeMode.NO_BRAKE;
    Main.M1.nEnableMode := ENUM_StageEnableMode.DURING_MOTION;
    END_IF

fb_MC_Y(stMotionStage := Main.M1);

END_PROGRAM

// ---- POUs/PRG_GasJetPointing.TcPOU
PROGRAM PRG_GasJetPointing
VAR
    fb_GSJP_X : FB_MotionStage;
    fb_GSJP_Z : FB_MotionStage;
    bInit : BOOL := TRUE;
END_VAR

IF ( bInit) THEN
    bInit := FALSE;
    Main.M4.bHardwareEnable := TRUE;
    Main.M4.bPowerSelf := TRUE;
    Main.M4.nBrakeMode := ENUM_StageBrakeMode.NO_BRAKE;
    Main.M4.nEnableMode := ENUM_StageEnableMode.DURING_MOTION;

    Main.M5.bHardwareEnable:= TRUE;
    Main.M5.bPowerSelf := TRUE;
    Main.M5.nBrakeMode := ENUM_StageBrakeMode.NO_BRAKE;
    Main.M5.nEnableMode := ENUM_StageEnableMode.DURING_MOTION;
    END_IF

fb_GSJP_X(stMotionStage := Main.M4);
fb_GSJP_Z(stMotionStage := Main.M5);

END_PROGRAM

// ---- POUs/PRG_CoilMovers.TcPOU
PROGRAM PRG_CoilMovers
VAR
    fb_Coil_Yaw : FB_MotionStage;
    fb_Coil_Roll : FB_MotionStage;
    bInit : BOOL := TRUE;
END_VAR


IF ( bInit) THEN
    bInit := FALSE;
    Main.M2.bHardwareEnable := TRUE;
    Main.M2.bPowerSelf := TRUE;
    Main.M2.nBrakeMode := ENUM_StageBrakeMode.NO_BRAKE;
    Main.M2.nEnableMode := ENUM_StageEnableMode.DURING_MOTION;

    Main.M3.bHardwareEnable:= TRUE;
    Main.M3.bPowerSelf := TRUE;
    Main.M3.nBrakeMode := ENUM_StageBrakeMode.NO_BRAKE;
    Main.M3.nEnableMode := ENUM_StageEnableMode.DURING_MOTION;
END_IF

Main.M2.bLimitForwardEnable := NOT Main.M2.bLimitForwardEnable;
Main.M2.bLimitBackwardEnable := NOT Main.M2.bLimitBackwardEnable;
fb_Coil_Roll(stMotionStage := Main.M2);

Main.M3.bLimitForwardEnable := NOT Main.M3.bLimitForwardEnable;
Main.M3.bLimitBackwardEnable := NOT Main.M3.bLimitBackwardEnable;
fb_Coil_Yaw(stMotionStage := Main.M3);

END_PROGRAM

// ---- POUs/PRG_SMARACT.TcPOU
PROGRAM PRG_SMARACT
VAR
    (*
    {attribute 'TcLinkToOSO' := '
        .stDS402Drive.nModeOfOperationNC	:=<0,8,0>TINC^NC-Task 1^Axes^M9_DREAM_DGPD_MMT_Y^Drive^Outputs^Out^nCtrl5;
        .stDS402Drive.nDS402DriveControlNC := <0,8,0>TINC^NC-Task 1^Axes^M9_DREAM_DGPD_MMT_Y^Drive^Outputs^Out^nCtrl1;
        .stDS402Drive.nDS402DriveControlNC := <8,8,0>TINC^NC-Task 1^Axes^M9_DREAM_DGPD_MMT_Y^Drive^Outputs^Out^nCtrl2
    '}
    {attribute 'TcLinkTo' := '
        .stDS402Drive.nSlaveAddr:=TIID^Device 1 (EtherCAT)^B940_009_R19_DRL_02_E0_EK1200^R19_DRL_02_E4_EK1122^TMO-DREAM-SMARACT-03^InfoData^AdsAddr^port;
        .stDS402Drive.stDS402DriveStatus:=TIID^Device 1 (EtherCAT)^B940_009_R19_DRL_02_E0_EK1200^R19_DRL_02_E4_EK1122^TMO-DREAM-SMARACT-03^DREAM:DGPD:MMT:Y^mode/status/pos/fError TxPDO^Status Word;
        .stDS402Drive.nFollowingError:=;TIID^Device 1 (EtherCAT)^B940_009_R19_DRL_02_E0_EK1200^R19_DRL_02_E4_EK1122^TMO-DREAM-SMARACT-03^DREAM:DGPD:MMT:Y^mode/status/pos/fError TxPDO^Following Error Actual Value;
        .stDS402Drive.nModeOfOperation:=TIID^Device 1 (EtherCAT)^B940_009_R19_DRL_02_E0_EK1200^R19_DRL_02_E4_EK1122^TMO-DREAM-SMARACT-03^DREAM:DGPD:MMT:Y^ctl/mode/pos RxPDO^Modes of Operation;
        .stDS402Drive.nModeOfOperationDisplay:=TIID^Device 1 (EtherCAT)^B940_009_R19_DRL_02_E0_EK1200^R19_DRL_02_E4_EK1122^TMO-DREAM-SMARACT-03^DREAM:DGPD:MMT:Y^mode/status/pos/fError TxPDO^Modes of Operation Display;
        .stDS402Drive.nDS402DriveControl:=TIID^Device 1 (EtherCAT)^B940_009_R19_DRL_02_E0_EK1200^R19_DRL_02_E4_EK1122^TMO-DREAM-SMARACT-03^DREAM:DGPD:MMT:Y^ctl/mode/pos RxPDO^Control Word
    '}
    fb_DGPD_Y : FB_MotionStageMCS2CSP ( stPiezoStage:=Main.M9, eModule:=E_Module.CHAN1 );
         {attribute 'TcLinkToOSO' := '
        .stDS402Drive.nModeOfOperationNC	:=<0,8,0>TINC^NC-Task 1^Axes^M10_DREAM_DGPD_MMT_X^Drive^Outputs^Out^nCtrl5;
        .stDS402Drive.nDS402DriveControlNC := <0,8,0>TINC^NC-Task 1^Axes^M10_DREAM_DGPD_MMT_X^Drive^Outputs^Out^nCtrl1;
        .stDS402Drive.nDS402DriveControlNC := <8,8,0>TINC^NC-Task 1^Axes^M10_DREAM_DGPD_MMT_X^Drive^Outputs^Out^nCtrl2
    '}
    {attribute 'TcLinkTo' := '
        .stDS402Drive.nSlaveAddr:=TIID^Device 1 (EtherCAT)^B940_009_R19_DRL_02_E0_EK1200^R19_DRL_02_E4_EK1122^TMO-DREAM-SMARACT-03^InfoData^AdsAddr^port;
        .stDS402Drive.stDS402DriveStatus:=TIID^Device 1 (EtherCAT)^B940_009_R19_DRL_02_E0_EK1200^R19_DRL_02_E4_EK1122^TMO-DREAM-SMARACT-03^DREAM:DGPD:MMT:X^mode/status/pos/fError TxPDO^Status Word;
        .stDS402Drive.nFollowingError:=TIID^Device 1 (EtherCAT)^B940_009_R19_DRL_02_E0_EK1200^R19_DRL_02_E4_EK1122^TMO-DREAM-SMARACT-03^DREAM:DGPD:MMT:X^mode/status/pos/fError TxPDO^Following Error Actual Value;
        .stDS402Drive.nModeOfOperation:=TIID^Device 1 (EtherCAT)^B940_009_R19_DRL_02_E0_EK1200^R19_DRL_02_E4_EK1122^TMO-DREAM-SMARACT-03^DREAM:DGPD:MMT:X^ctl/mode/pos RxPDO^Modes of Operation;
        .stDS402Drive.nModeOfOperationDisplay:=TIID^Device 1 (EtherCAT)^B940_009_R19_DRL_02_E0_EK1200^R19_DRL_02_E4_EK1122^TMO-DREAM-SMARACT-03^DREAM:DGPD:MMT:X^mode/status/pos/fError TxPDO^Modes of Operation Display;
        .stDS402Drive.nDS402DriveControl:=TIID^Device 1 (EtherCAT)^B940_009_R19_DRL_02_E0_EK1200^R19_DRL_02_E4_EK1122^TMO-DREAM-SMARACT-03^DREAM:DGPD:MMT:X^ctl/mode/pos RxPDO^Control Word
    '}
    fb_DGPD_X : FB_MotionStageMCS2CSP ( stPiezoStage:=Main.M10, eModule:=E_Module.CHAN2 );
       {attribute 'TcLinkToOSO' := '
        .stDS402Drive.nModeOfOperationNC	:=<0,8,0>TINC^NC-Task 1^Axes^M11_DREAM_DGPD_MMT_RET^Drive^Outputs^Out^nCtrl5;
        .stDS402Drive.nDS402DriveControlNC := <0,8,0>TINC^NC-Task 1^Axes^M11_DREAM_DGPD_MMT_RET^Drive^Outputs^Out^nCtrl1;
        .stDS402Drive.nDS402DriveControlNC := <8,8,0>TINC^NC-Task 1^Axes^M11_DREAM_DGPD_MMT_RET^Drive^Outputs^Out^nCtrl2
    '}
    {attribute 'TcLinkTo' := '
        .stDS402Drive.nSlaveAddr:=TIID^Device 1 (EtherCAT)^B940_009_R19_DRL_02_E0_EK1200^R19_DRL_02_E4_EK1122^TMO-DREAM-SMARACT-03^InfoData^AdsAddr^port;
        .stDS402Drive.stDS402DriveStatus:=TIID^Device 1 (EtherCAT)^B940_009_R19_DRL_02_E0_EK1200^R19_DRL_02_E4_EK1122^TMO-DREAM-SMARACT-03^DREAM:DGPD:MMT:RET^mode/status/pos/fError TxPDO^Status Word;
        .stDS402Drive.nFollowingError:=TIID^Device 1 (EtherCAT)^B940_009_R19_DRL_02_E0_EK1200^R19_DRL_02_E4_EK1122^TMO-DREAM-SMARACT-03^DREAM:DGPD:MMT:RET^mode/status/pos/fError TxPDO^Following Error Actual Value;
        .stDS402Drive.nModeOfOperation:=TIID^Device 1 (EtherCAT)^B940_009_R19_DRL_02_E0_EK1200^R19_DRL_02_E4_EK1122^TMO-DREAM-SMARACT-03^DREAM:DGPD:MMT:RET^ctl/mode/pos RxPDO^Modes of Operation;
        .stDS402Drive.nModeOfOperationDisplay:=TIID^Device 1 (EtherCAT)^B940_009_R19_DRL_02_E0_EK1200^R19_DRL_02_E4_EK1122^TMO-DREAM-SMARACT-03^DREAM:DGPD:MMT:RET^mode/status/pos/fError TxPDO^Modes of Operation Display;
        .stDS402Drive.nDS402DriveControl:=TIID^Device 1 (EtherCAT)^B940_009_R19_DRL_02_E0_EK1200^R19_DRL_02_E4_EK1122^TMO-DREAM-SMARACT-03^DREAM:DGPD:MMT:RET^ctl/mode/pos RxPDO^Control Word
    '}
    fb_DGPD_RET : FB_MotionStageMCS2CSP ( stPiezoStage:=Main.M11, eModule:=E_Module.CHAN3 );

    stDGPD_RET: ARRAY[1..GeneralConstants.MAX_STATES] OF ST_PositionState;

    {attribute 'pytmc' := '
          pv: DGPD:RET:STATES:SET
          io: io
    '}
     stDGPD_RET_Set: ENUM_AxisStates;
        {attribute 'pytmc' := '
          pv: DGPD:RET:STATES:GET
          io: i
        '}
    stDGPD_RET_Get: ENUM_AxisStates;

    fbDGPD_RET_PMPStates: FB_PositionStatePMPS1D;
    *)
END_VAR

(*
fbDGPD_RET_PMPStates(
    stMotionStage:=Main.M11,
    astPositionState:=stDGPD_RET,
    eEnumSet:=stDGPD_RET_Set,
    eEnumGet:=stDGPD_RET_Get,
    sDeviceName := 'DREAM:DGPD:MMT:RET',
    sTransitionKey := 'DREAM:DGPD:MMT:RET-TRANSITION',
    fbFFHWO:=GVL_PMPS.fbFastFaultOutput1,
    fbArbiter:=GVL_PMPS.fbArbiter1,
    bEnableMotion:=TRUE,
    bEnableBeamParams:=TRUE,
    bEnablePositionLimits:=TRUE,
    bReadDBNow:=TRUE,
);

fb_DGPD_RET();
fb_DGPD_X();
fb_DGPD_Y();
*)

END_PROGRAM
